// TIA Portal V19 export
TYPE "C215_VAR_IF_SVLU_TYPIC"
   STRUCT
      STS_UIT { ExternalAccessible := 'False'; ExternalVisible := 'False'; ExternalWritable := 'False'} : Bool;   // Statisch indicatiebord vluchtroute uit
      EXT_AUT { ExternalAccessible := 'False'; ExternalVisible := 'False'; ExternalWritable := 'False'} : Bool;   // Externe (hoofd) beveiliging aangesproken
      EXT_HW { ExternalAccessible := 'False'; ExternalVisible := 'False'; ExternalWritable := 'False'} : Bool;   // Sturings hardware (PLC) in storing
      STO { ExternalAccessible := 'False'; ExternalVisible := 'False'; ExternalWritable := 'False'} : Struct   // Opsomming van alle storingen
         A001 : Bool;   // Beveiliging aangesproken
         AT01 : Bool;   // Foute terugmelding: Indicatiebord uitgestuurd, terugmelding Uit niet (of te laat) ontvangen
         AT02 : Bool;   // Foute terugmelding: Indicatiebord niet uitgestuurd, terugmelding Uit blijft aanwezig
      END_STRUCT;
   END_STRUCT;
END_TYPE
